# EPICS alarm handler configuration: mps_database/bareTest/alarms/areas/mpln_l2b_mp02.alhConfig
GROUP NULL MPLN:L2B:MP02:1
$ALIAS MPS Link Node 61
$GUIDANCE
LTUH MPS
   Group Name: MPLN:L2B:MP02:1
   Summary PV:  MPLN:L2B:MP02:1:STATSUMY
$END
CHANNEL  MPLN:L2B:MP02:1    MPLN:L2B:MP02:1:MPS_EN_RBV		-----
CHANNEL  MPLN:L2B:MP02:1    MPLN:L2B:MP02:1:LC1_MODE_RBV		-----
